// TIA Portal V20 export
DATA_BLOCK "DB_Manual"   // DB18
// stored: Access Published, MemoryReserve 100, Namespace EmptyLine
   VAR
      Conveyor : Struct
         ID : Int;
         Enable : Bool;
         Run : Bool;
         in : Bool;
      END_STRUCT;
      Line : Struct
         EmptyLine : Struct
            Conveyor { S7_SetPoint := 'True'} : Array[_.minEmptyLine.._.maxEmptyLine] of "Global.ManualInputs";
         END_STRUCT;
      END_STRUCT;
   END_VAR
BEGIN
END_DATA_BLOCK
